PROGRAM MAIN
VAR
END_VAR

P_Safety();
P_Alarm();
P_Patlite();
P_BasicMotion();
P_WriteMotion();
P_MitsubishiCommunication();

END_PROGRAM

(* stored: Version 1.1.0.1, ProductVersion 3.1.4024.12
   POU MAIN: Id {50158451-d374-4957-970b-65b4e1d88bf2}, SpecialFunc None *)
